FUNCTION_BLOCK VSG_OperatingModes_alt
VAR_INPUT
	Start 			: BOOL;
	Stop			: BOOL;
	Reset			: BOOL;
	Schalter		: BOOL;
	Schrittkette_GS : BOOL;
END_VAR
VAR_OUTPUT
	A1 : BOOL; //Initialzustand
	A2 : BOOL; //Stillstand angefordert am Ende des Zyklus
//	A3 : BOOL; //Stillstand angefordert in einem bestimmten Zustand
//	A4 : BOOL; //Erhaltener Stillstand
//	A5 : BOOL; //Vorbereitung zur Wiederaufnahme nach Störung
	A6 : BOOL; //Fahrt in den Initialzustand
	F1 : BOOL; //Normalbetrieb
//	F2 : BOOL; //Anfahren
//	F3 : BOOL; //Abfahren
	F4 : BOOL; //Handbetrieb
//	F5 : BOOL; //Schrittbetrieb
//	F6 : BOOL; //Testbetrieb
//	D1 : BOOL; //Not-Aus
//	D2 : BOOL; //DIagnose und Störbehandlung
//	D3 : BOOL; //Produktion trotz Störung
END_VAR
VAR
	bFirstScan : BOOL := TRUE;	
	
	RS_InitialState: RS;	
	RS_InitialDrive: RS;
	RS_ManualOperationMode: RS;
	RS_AutomaticOperationMode: RS;
	RS_CycleEnded: RS;

	R_TRIG_Manual: R_TRIG;
	R_TRIG_Automatic: R_TRIG;
	R_TRIG_InitialDrive: R_TRIG;
	R_TRIG_CycleEnded: R_TRIG;
	R_TRIG_Init: R_TRIG;
END_VAR
VAR // added by the converter: edge detectors and wires of the graphical bodies
    _w1 : BOOL;
END_VAR

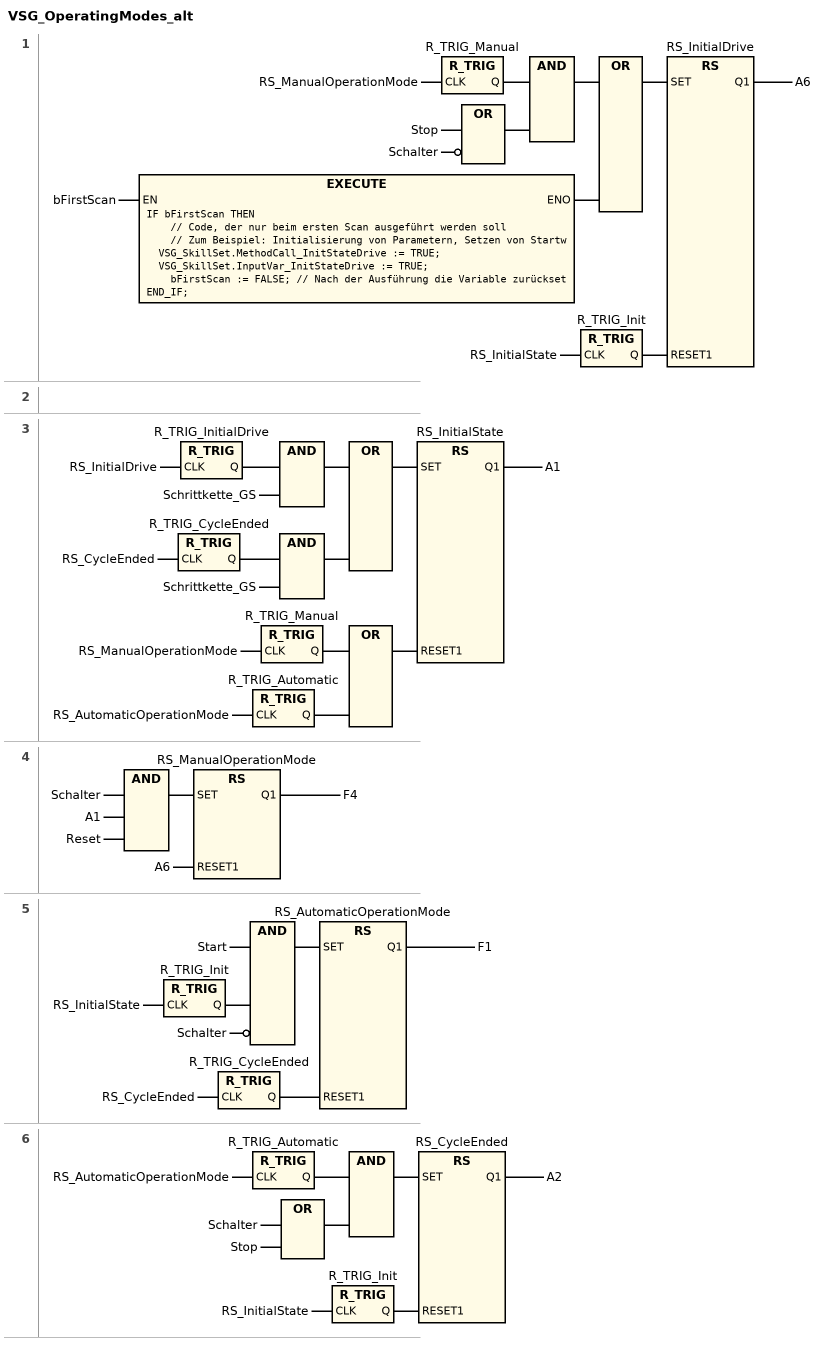
// NETWORK 1
R_TRIG_Manual(CLK := RS_ManualOperationMode); // R_TRIG
_w1 := bFirstScan;
IF _w1 THEN
    IF bFirstScan THEN
        // Code, der nur beim ersten Scan ausgeführt werden soll
        // Zum Beispiel: Initialisierung von Parametern, Setzen von Startwerten etc.
    	VSG_SkillSet.MethodCall_InitStateDrive := TRUE;
    	VSG_SkillSet.InputVar_InitStateDrive := TRUE;
        bFirstScan := FALSE; // Nach der Ausführung die Variable zurücksetzen
    END_IF;
END_IF
R_TRIG_Init(CLK := RS_InitialState); // R_TRIG
RS_InitialDrive(SET := R_TRIG_Manual.Q AND (Stop OR NOT Schalter) OR _w1, RESET1 := R_TRIG_Init.Q); // RS
A6 := RS_InitialDrive.Q1;

// NETWORK 2

// NETWORK 3
R_TRIG_InitialDrive(CLK := RS_InitialDrive); // R_TRIG
R_TRIG_CycleEnded(CLK := RS_CycleEnded); // R_TRIG
R_TRIG_Manual(CLK := RS_ManualOperationMode); // R_TRIG
R_TRIG_Automatic(CLK := RS_AutomaticOperationMode); // R_TRIG
RS_InitialState(SET := R_TRIG_InitialDrive.Q AND Schrittkette_GS OR R_TRIG_CycleEnded.Q AND Schrittkette_GS, RESET1 := R_TRIG_Manual.Q OR R_TRIG_Automatic.Q); // RS
A1 := RS_InitialState.Q1;

// NETWORK 4
RS_ManualOperationMode(SET := Schalter AND A1 AND Reset, RESET1 := A6); // RS
F4 := RS_ManualOperationMode.Q1;

// NETWORK 5
R_TRIG_Init(CLK := RS_InitialState); // R_TRIG
R_TRIG_CycleEnded(CLK := RS_CycleEnded); // R_TRIG
RS_AutomaticOperationMode(SET := Start AND R_TRIG_Init.Q AND NOT Schalter, RESET1 := R_TRIG_CycleEnded.Q); // RS
F1 := RS_AutomaticOperationMode.Q1;

// NETWORK 6
R_TRIG_Automatic(CLK := RS_AutomaticOperationMode); // R_TRIG
R_TRIG_Init(CLK := RS_InitialState); // R_TRIG
RS_CycleEnded(SET := R_TRIG_Automatic.Q AND (Schalter OR Stop), RESET1 := R_TRIG_Init.Q); // RS
A2 := RS_CycleEnded.Q1;

END_FUNCTION_BLOCK

(* stored: Version 1.1.0.1, ProductVersion 3.1.4026.18
   POU VSG_OperatingModes_alt: Id {8394f1d5-fe9e-48c9-a63e-e5fd3f29b475}, SpecialFunc None *)
